{attribute 'GeneratedUsingTerminal: EL2596-0000-0017'}
{attribute addProperty BoxType "EL2596-0000-0017"}
{attribute addProperty Id "ControlAT %Q*Control_12F99C765"}
{attribute addProperty CRC "2979117971"}
{attribute addProperty Size "5"}
TYPE DOX_Control_B191BB93 EXTENDS OutputBase_10CEE7DE :
STRUCT
	{attribute addProperty Name "Control"}
	Control AT %Q* : Control_12F99C76;
END_STRUCT
END_TYPE

(* stored: Version 1.2.0.0, ProductVersion 3.1.4024.11
   DUT DOX_Control_B191BB93: Id {863f6bd3-410f-4d89-9aef-d9f85c1efbc9} *)
